// Mitsubishi GX Works2 project: XOR   PLC: Q03UDV

PROGRAM MAIN
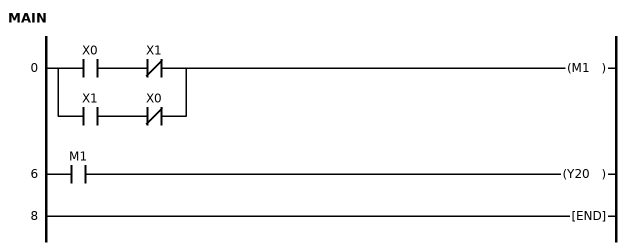
0     LD      X0
      ANI     X1
      LD      X1
      ANI     X0
      ORB
      OUT     M1
6     LD      M1
      OUT     Y20
8     END
END_PROGRAM
